Yaskawa INFORM job: R1_W28-29-A1(180,180)KM-OK.JBI

/JOB
//NAME R1_W28-29-A1(180,180)KM-OK
///FOLDERNAME KRIS-SCIANA
//POS
///NPOS 65,65,0,3,0,0
///TOOL 0
///POSTYPE PULSE
///PULSE
C00000=-67773,-115242,-103906,-19623,25601,63975
C00001=-3416,-115242,-103906,-19623,25601,63975
C00002=-26455,-158011,-118219,-7266,71058,46254
C00003=-3769,-166785,-97381,-40477,88405,55422
C00004=-43833,-163320,-90260,-51767,68136,47699
C00005=-58180,-159732,-87945,-54234,61162,44648
C00006=-63603,-157963,-86981,-54851,58553,43409
C00007=-66278,-157921,-85919,-55509,56788,43136
C00008=-63603,-157963,-86981,-54851,58553,43409
C00009=-65450,-156876,-86867,-54833,57883,42815
C00010=-52071,-149058,-81923,-55655,69408,45894
C00011=-46903,-150011,-82682,-54556,72120,46872
C00012=-33933,-151550,-84471,-51325,78972,49252
C00013=745,-148481,-92489,-40496,100018,54785
C00014=745,-148481,-92489,-40496,100018,-31489
C00015=2942,-154737,-74876,-64026,90754,-45137
C00016=-12687,-153905,-71509,-70780,81542,-46215
C00017=-26655,-152993,-68740,-76840,73348,-46850
C00018=-30120,-152698,-68741,-78234,71425,-47160
C00019=-20060,-153266,-70138,-73933,77260,-46662
C00020=-2668,-108271,-36394,-73800,106169,-49661
C00021=-2795,-109689,-36612,-73668,105914,-49396
C00022=-2668,-108271,-36394,-73800,106169,-49661
C00023=-11616,-151136,-71396,-66783,83877,-47366
C00024=-32155,-152631,-71044,-75120,72021,-48974
C00025=-32155,-151654,-70089,-75145,71998,-48934
C00026=-27863,-153509,-71457,-73490,74398,-48519
C00027=-11616,-151136,-71396,-66783,83877,-47366
C00028=-25506,-151332,-72561,-72163,76318,-49113
C00029=-19601,-151946,-73933,-69823,79872,-48749
C00030=-6609,-152805,-77281,-64652,87841,-47902
C00031=11727,-148546,-70447,-67430,88261,-26161
C00032=-2786,-144833,-66398,-73418,79847,-27384
C00033=-7846,-143581,-65196,-75440,76898,-27767
C00034=-2740,-143069,-64570,-73432,79805,-27283
C00035=-8600,-144897,-66597,-75699,76514,-27912
C00036=-8494,-143668,-65314,-75685,76528,-27832
C00037=-8383,-143667,-65311,-75641,76593,-27822
C00038=-8691,-143206,-65104,-75745,76446,-27896
C00039=-2512,-144864,-66427,-73308,80004,-27361
C00040=11995,-148561,-70475,-67317,88414,-26135
C00041=-5762,-130033,-61860,-71470,91120,-47000
C00042=-16585,-122609,-65225,-67002,86845,-63997
C00043=-9171,-129764,-63022,-72784,89349,-47711
C00044=-5520,-130035,-61860,-71377,91265,-46975
C00045=-6742,-110566,-55810,-71091,90544,-52668
C00046=-11835,-150105,-78679,-69823,68177,-44206
C00047=1775,-179748,-92792,-71004,87182,-59781
C00048=7163,-163778,-82041,-73169,95228,-78609
C00049=3601,-158687,-77326,-74749,93097,-78785
C00050=-7911,-173992,-90877,-73988,81334,-63025
C00051=-1337,-176331,-90920,-71361,84686,-61910
C00052=4961,-150498,-69477,-74074,93688,-78395
C00053=5073,-140061,-58180,-73752,92660,-76555
C00054=-4182,-142299,-62269,-72072,85812,-79389
C00055=296,-170101,-89745,-70135,89267,-80092
C00056=296,-183640,-100514,-70129,89146,-79949
C00057=296,-177280,-100514,-70129,56506,-79949
C00058=-225,-181834,-128144,-48952,36574,-78492
C00059=-253,-180984,-127857,-3714,35873,-78525
C00060=-253,-180984,-127857,-3714,2349,-78525
C00061=-253,-180984,-127857,-3714,-15943,-78525
C00062=-253,-184426,-130262,-3650,-16231,-78554
C00063=-298,-184426,-130262,-3650,-16231,-78554
C00064=-105101,-184426,-130262,-3650,-16231,-78554
BC00000=395863,1065,1067434
BC00001=63554,1065,1067434
BC00002=141105,738,1069846
BC00003=170623,15,1075175
BC00004=170623,15,1075175
BC00005=170623,15,1075175
BC00006=170623,15,1075175
BC00007=170622,15,1075171
BC00008=170623,15,1075175
BC00009=170623,15,1075175
BC00010=170623,15,1075175
BC00011=170623,15,1075175
BC00012=170623,15,1075175
BC00013=180341,15,1075175
BC00014=180341,15,1075175
BC00015=201429,15,1062136
BC00016=201429,15,1062136
BC00017=201429,15,1062136
BC00018=201429,15,1062136
BC00019=201429,15,1062136
BC00020=201429,15,1062136
BC00021=201429,15,1062136
BC00022=201429,15,1062136
BC00023=201429,15,1062136
BC00024=201429,15,1062136
BC00025=201429,15,1062136
BC00026=201429,15,1062136
BC00027=201429,15,1062136
BC00028=201429,15,1062136
BC00029=201429,15,1062136
BC00030=201429,15,1062136
BC00031=168347,15,1075175
BC00032=167620,15,1075175
BC00033=167329,15,1075175
BC00034=167329,15,1075175
BC00035=167329,15,1075175
BC00036=162551,15,1075175
BC00037=138184,15,1075175
BC00038=133405,15,1075175
BC00039=133696,15,1075175
BC00040=134423,15,1075175
BC00041=142471,15,1070365
BC00042=136010,15,1075175
BC00043=140896,15,1064894
BC00044=140896,15,1064894
BC00045=121757,15,1075175
BC00046=122355,15,1075175
BC00047=193001,15,921179
BC00048=190996,15,924583
BC00049=190996,15,924583
BC00050=190996,15,924590
BC00051=190996,15,924590
BC00052=190996,15,924583
BC00053=190996,15,924583
BC00054=190996,15,924583
BC00055=190997,15,924582
BC00056=190997,15,924582
BC00057=190997,15,924582
BC00058=91599,16,924574
BC00059=91535,16,924574
BC00060=91535,16,924574
BC00061=91535,16,924574
BC00062=88712,16,1053735
BC00063=390854,16,1053735
BC00064=390854,16,1053735
///POSTYPE BASE
///RECTAN
///RCONF 0,0,0,0,1,0,0,0,0,0,0,0,0,0,0,0,0,0,0,0,0,0,0,0
P00006=2.006,1.622,-0.565,0.0000,0.0000,0.0000
P00022=2.006,1.622,-0.565,0.0000,0.0000,0.0000
///RCONF 0,0,0,0,0,0,0,0,0,0,0,0,0,0,0,0,0,0,0,0,0,0,0,0
P00023=-2.957,-4.083,2.762,0.0000,0.0000,0.0000
//INST
///DATE 2023/11/29 20:07
///ATTR SC,RW
///GROUP1 RB1,BS1
NOP
'r1_W28-29-A1(180,180)
'Path S1019
SFTOF
MOVJ C00000 BC00000 VJ=20.00
MOVJ C00001 BC00001 VJ=20.00
MOVJ C00002 BC00002 VJ=20.00
MOVJ C00003 BC00003 VJ=20.00
MOVL C00004 BC00004 V=166.7
MOVL C00005 BC00005 V=166.7
MOVL C00006 BC00006 V=60.0
REFP 3 C00007 BC00007
CALL JOB:SEARCH-R1
SET P023 P006
SFTON P023
MOVL C00008 BC00008 V=60.0
REFP 3 C00009 BC00009
CALL JOB:SEARCH-R1
SET P023 P006
SFTON P023
MOVL C00010 BC00010 V=60.0
MOVL C00011 BC00011 V=100.0
MOVL C00012 BC00012 V=166.7
'Path VIA1135
SFTOF
MOVJ C00013 BC00013 VJ=20.00
'Path VIA1136
SFTOF
MOVJ C00014 BC00014 VJ=20.00
'Path S1020
SFTOF
MOVJ C00015 BC00015 VJ=20.00
MOVJ C00016 BC00016 VJ=20.00
MOVL C00017 BC00017 V=60.0
REFP 3 C00018 BC00018
CALL JOB:SEARCH-R1
SET P022 P006
SFTON P022
MOVL C00019 BC00019 V=60.0
MOVL C00020 BC00020 V=60.0
REFP 3 C00021 BC00021
CALL JOB:SEARCH-R1
SET P022 P006
SFTON P022
MOVL C00022 BC00022 V=60.0
MOVL C00023 BC00023 V=100.0
MOVL C00024 BC00024 V=60.0
REFP 3 C00025 BC00025
CALL JOB:SEARCH-R1
SET P022 P006
SFTON P022
MOVL C00026 BC00026 V=60.0
MOVL C00027 BC00027 V=100.0
MOVL C00028 BC00028 V=100.0
MOVL C00029 BC00029 V=100.0
MOVL C00030 BC00030 V=166.7
'Path W1021
SFTOF
SFTON P022
MOVJ C00031 BC00031 VJ=20.00
MOVJ C00032 BC00032 VJ=20.00
MOVL C00033 BC00033 V=100.0 PL=0
REFP 1 C00034 BC00034
REFP 2 C00035 BC00035
MACRO1 MJ#(0) ARGF9
ARCON
MOVL C00036 BC00036 V=10.8
MOVL C00037 BC00037 V=10.8
MOVL C00038 BC00038 V=10.8
ARCOF
MOVL C00039 BC00039 V=100.0
MOVL C00040 BC00040 V=166.7
SFTOF
'Path W1022
SFTOF
SFTON P023
MOVL C00041 BC00041 V=100.0
MOVL C00042 BC00042 V=100.0 PL=0
REFP 1 C00043 BC00043
REFP 2 C00044 BC00044
MACRO1 MJ#(0) ARGF7
ARCON
MOVL C00045 BC00045 V=10.0
ARCOF
MOVL C00046 BC00046 V=100.0
SFTOF
'Path W1023
SFTOF
SFTON P022
MOVL C00047 BC00047 V=100.0
MOVL C00048 BC00048 V=100.0
MOVL C00049 BC00049 V=100.0 PL=0
REFP 1 C00050 BC00050
REFP 2 C00051 BC00051
MACRO1 MJ#(0) ARGF7
ARCON
MOVL C00052 BC00052 V=10.0
MOVL C00053 BC00053 V=10.0
MOVL C00054 BC00054 V=10.0
ARCOF
MOVL C00055 BC00055 V=100.0
SFTOF
MOVL C00056 BC00056 V=100.0
MOVL C00057 BC00057 V=100.0
MOVL C00058 BC00058 V=100.0
MOVL C00059 BC00059 V=100.0
MOVL C00060 BC00060 V=100.0
SFTOF
MOVL C00061 BC00061 V=100.0
MOVJ C00062 BC00062 VJ=20.00
MOVJ C00063 BC00063 VJ=20.00
MOVJ C00064 BC00064 VJ=20.00
END
